(* PLC project Unnamed, Unknown Unnamed 1 *)
(* stored: creationDateTime 2026-10-02T14:32:02, modificationDateTime 2026-10-02T22:33:47 *)

PROGRAM program0
  VAR
    TankFillAuto_Cmd : BOOL;  (* Internal automatic fill latch/command *)
    TankValveOpen : BOOL;  (* Discrete command/status for the fill valve *)
    EStop_Cmd : BOOL;  (* Emergency-stop input; TRUE forces automatic fill to stop *)
    TankLevelHi_Alarm : BOOL;  (* High-level alarm state *)
    TankLevelLo_Alarm : BOOL;  (* Low-level alarm state *)
  END_VAR
  VAR_INPUT
    TankLevel_LIT : REAL := 0.5 ft;  (* Measured tank level in feet *)
    TankEmpty_SP : REAL := 2.0ft;  (* Automatic fill start setpoint (2.0 ft) *)
    TankFull_SP : REAL := 8.0ft;  (* Automatic fill stop setpoint (8.0 ft) *)
  END_VAR
  VAR
    TankLevelHi_Alarm_SP : BOOL := 9.0ft;  (* High-level alarm setpoint (9.0 ft) *)
    TankLevelLoAlarm_SP : BOOL := 1.0ft;  (* Low-level alarm setpoint (1.0 ft) *)
  END_VAR

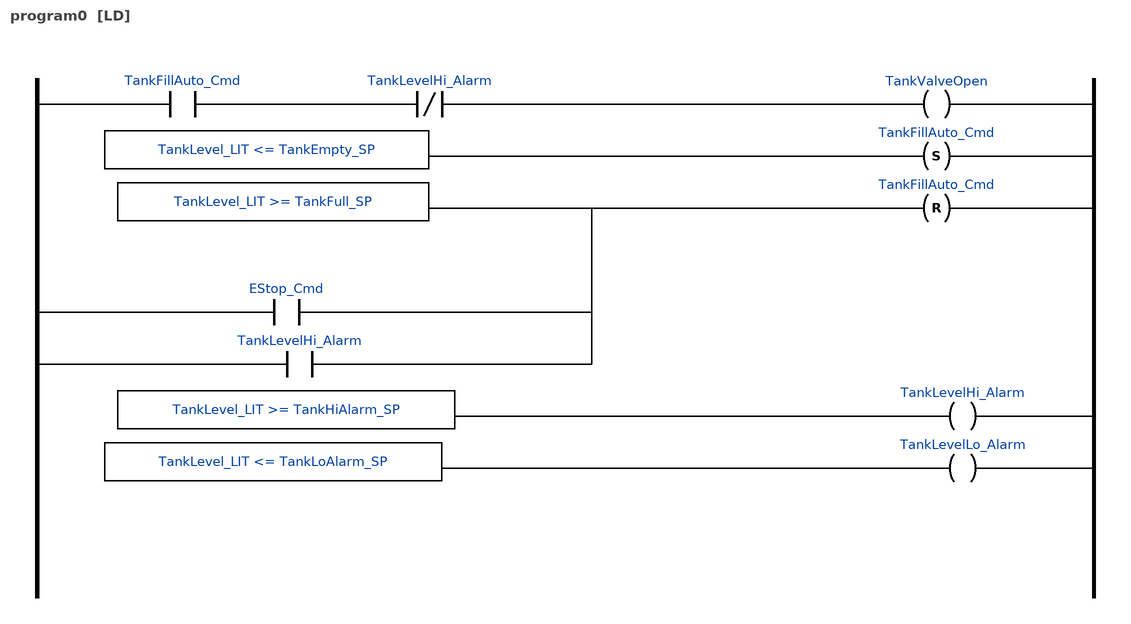
(* LD diagram, written out as Structured Text *)
TankValveOpen := TankFillAuto_Cmd AND NOT TankLevelHi_Alarm;
IF TankLevel_LIT <= TankEmpty_SP THEN TankFillAuto_Cmd := TRUE; END_IF;
IF (TankLevel_LIT >= TankFull_SP) OR EStop_Cmd OR TankLevelHi_Alarm THEN TankFillAuto_Cmd := FALSE; END_IF;
TankLevelHi_Alarm := TankLevel_LIT >= TankHiAlarm_SP;
TankLevelLo_Alarm := TankLevel_LIT <= TankLoAlarm_SP;
END_PROGRAM

CONFIGURATION Config0
  RESOURCE Res0 ON PLC
    TASK task0(INTERVAL := T#20ms, PRIORITY := 0);
    PROGRAM instance0 WITH task0 : program0;
  END_RESOURCE
END_CONFIGURATION
